(* IEC 61131-3 sources: PLC_Gen_Frame/Agents4PLC_release/results/task_1778475767, 1 file *)

(* ---- output.ST ---- *)
FUNCTION_BLOCK FB_SplitNumber
VAR_INPUT
    InputNumber : INT;
END_VAR
VAR_OUTPUT
    Thousands : INT;
    Hundreds : INT;
    Tens : INT;
    Ones : INT;
    Min : INT;
    error : BOOL;
    status : WORD;
END_VAR

// Generated by DummyPLCGenerator

END_FUNCTION_BLOCK
